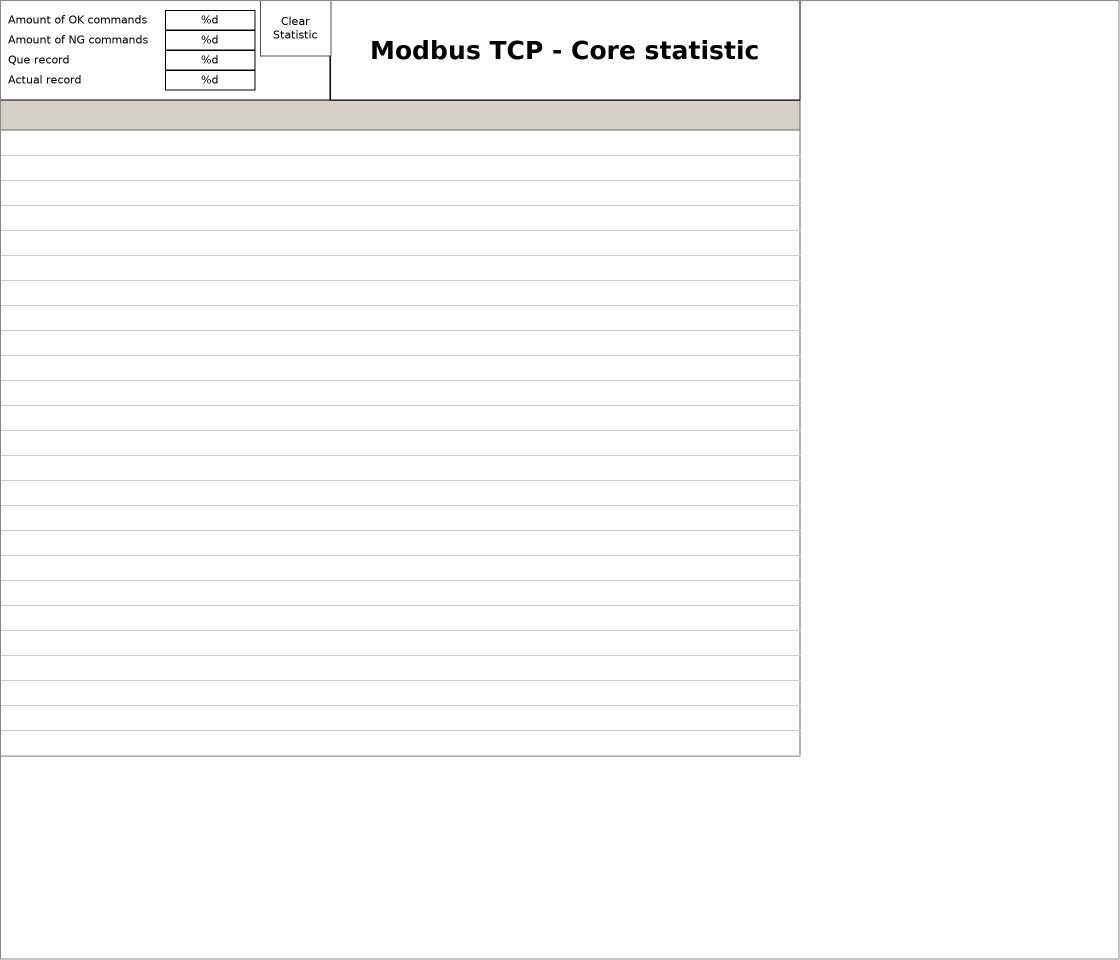
VISUALIZATION vModbusTcpCore  // 1120x960
VAR_IN_OUT
	stData : stModTcpCore_HmiData;
END_VAR
    Rectangle (0,0 330x100)
    Label (5,30 156x20), "Amount of NG commands"
    Rectangle (165,10 90x20), "%d", text variable: stData.iAmoutOfPerformedCommunications
    Label (5,10 166x20), "Amount of OK commands"
    Label (5,50 150x20), "Que record"
    Label (5,70 150x20), "Actual record"
    Rectangle (165,30 90x20), "%d", text variable: stData.iAmoutOfErrors
    Rectangle (165,50 90x20), "%d", text variable: stData.iLastQue
    Rectangle (165,70 90x20), "%d", text variable: stData.iActualQue
    Table (0,100 800x656), data array: stData.arVisuHist
        p1128707560: GVL_ModbusTCP_Constants.iCommuniactionHistoryLimit
        p3854506369: stData.arVisuHist[INDEX]
        p2232123230: IP | Identifier | Time | Communication Time | Error ID
    Rectangle (330,0 470x100), "Modbus TCP - Core statistic"
    Rectangle (260,0 71x56), "Clear Statistic"
        OnMouseClick: toggle stData.bClearStatistic
END_VISUALIZATION

(* stored: Version 1.1.0.1, ProductVersion 3.1.4024.13
   Visu vModbusTcpCore: Id {49f85ae8-ebfc-4e26-a597-92bbb4e3cbe4} *)
